TYPE F32 : REAL; END_TYPE

(* stored: Version 1.1.0.1
   DUT F32: Id {e6a27a94-241a-01ae-2161-3ed54fa5f617} *)
